FUNCTION "LAxisCtrl_UnpubSensorTypePosAxis" : DInt
{ S7_Optimized_Access := 'TRUE' }
AUTHOR : 'tech.team.motioncontrol@siemens.com'
FAMILY : AxisCtrl
VERSION : 1.1
   VAR_INPUT
      axis {InstructionName := 'TO_PositioningAxis'; LibVersion := '5.0'} : TO_PositioningAxis;
      index : Int;
   END_VAR


BEGIN
	// Read axis parameter
	#LAxisCtrl_UnpubSensorTypePosAxis := #axis.Sensor[#index].Type;
END_FUNCTION

